# EPICS SNL sequencer program: timingApp/src/timingSequence.st
program timingSequence ("T=,P=EVG1:,R=")

// Macros
//  T: Timing system record prefix.
//  P:, R: Event generator record prefixes.
// Defaults provided here can be overridden by seq command in st.cmd.

// No wait for connections
option -c;
// Safe mode
option +s;
// Enable run-time debug messages
option +d;

#include "timingSequenceConstants.h"
%%#include <stdio.h>
%%#include <stdlib.h>

/*
 * Additional ticks for end of cycle
 */
int endOfCycleDelay;
assign endOfCycleDelay to "{T}TimCycleDelay";
monitor endOfCycleDelay;

/*
 * Injection request waveform.
 */
int request[7];
assign request to "{T}TimInjReq";
monitor request;
evflag requestFlag;
sync request requestFlag;
unsigned int modeIndexes[255];
%{
typedef enum { /* Request waveform indices. */
        TARGET_BUCKET,
        GUN_BUNCHES,
        INJ_MODE,
        GUN_INHIBIT,
        TARGET_AR_BUCKET,
        FUTURE_USE_1,
        SEQUENCE,
} REQUEST_FIELDS;
}%

/* Values extracted from injection request waveform: */
int sequence = 0;       /* Sequence #: request ignored if no change from previous */
int lastSequence = -1;
int bucket = 1;         /* Target bucket (1-328) */
int arBucket = 1;       /* AR Target bucket (1-304) */
assign arBucket to "{T}TimTargetARBucket";
int bunches = 1;        /* Number of electron gun bunches (1-16) */
int inhibit = 0;        /* Inhibit electron gun if set, even if mode allows gun */
int mode = 0;           /* Type of injection sequence.  See eventListForMode() */
int injFieldSync = 0;   /* Injection field delay */
int extrFieldSync = 0;  /* Extraction field delay */
int extrFieldARSync = 0;  /* Extraction field AR delay */
int extrFieldARSyncSP = 0;  /* Extraction field AR delay in AR/BR alignment cycles */
int brTgtBucket = 1;  /* BR target bucket (in buckets) for AR injection */

int injFieldSyncDelay = 0;
assign injFieldSyncDelay to "{T}TimInjFieldSyncDelay";
monitor injFieldSyncDelay;
int extrFieldSyncDelay = 0;
assign extrFieldSyncDelay to "{T}TimExtrFieldSyncDelay";
monitor extrFieldSyncDelay;
int extrFieldARSyncDelay = 0;
assign extrFieldARSyncDelay to "{T}TimExtrFieldARSyncDelay";
monitor extrFieldARSyncDelay;
int extrFieldARSyncDelaySP = 0;
assign extrFieldARSyncDelaySP to "{T}TimExtrFieldARSyncDelaySP";
monitor extrFieldARSyncDelaySP;
int injStBRBucket = 1;
assign injStBRBucket to "{P}{R}INJ:stBRBucket";
monitor injStBRBucket;

/* Save value until we're ready to write to the FPGA */
int injSyncMode;
assign injSyncMode to "{T}TimInjSyncMode";
int injAlignSel;
assign injAlignSel to "{T}TimInjAlignSel";

/*
 * Monitor of injection request values sent to FPGA sequencer.
 */

int sequenceMon = 0;        /* Sequence #: request ignored if no change from previous */
assign sequenceMon to "{T}TimSequenceNumberMon";
int bucketMon = 1;          /* Target bucket (1-328) */
assign bucketMon to "{T}TimTargetBucketMon";
int arBucketMon = 1;          /* Target AR Bucket (1-304) */
assign arBucketMon to "{T}TimTargetARBucketMon";
int bunchesMon = 1;         /* Number of electron gun bunches (1-16) */
assign bunchesMon to "{T}TimGunBunchCountMon";
int inhibitMon = 0;         /* Inhibit electron gun if set, even if mode allows gun */
assign inhibitMon to "{T}TimGunInhibitMon";
int modeMon = 0;            /* Type of injection sequence.  See eventListForMode() */
assign modeMon to "{T}TimInjModeMon";
int injFieldSyncMon = 0;    /* Injection field delay */
assign injFieldSyncMon to "{T}TimInjFieldSyncDelayMon";
int extrFieldSyncMon = 0;   /* Extraction field delay */
assign extrFieldSyncMon to "{T}TimExtrFieldSyncDelayMon";
int extrFieldARSyncMon = 0;   /* Extraction field delay */
assign extrFieldARSyncMon to "{T}TimExtrFieldARSyncDelayMon";

/*
 * Calculated values
 */
int injStBRBucketIdx = 0;

int tgtBRDelayOffset = 0;
assign tgtBRDelayOffset to "{T}TimTgtBRDelayOffset";
int tgtBRBucket = 1;
assign tgtBRBucket to "{T}TimTgtBRBucket";

/*
 * Storage ring current.
 * Sequencer refuses to inject when this exceeds MAX_BEAM_CURRENT.
 */
double beamcurrent;
assign beamcurrent to "SR:DCCT:AVG";
monitor beamcurrent;

/*
 * Soft sequence timestamp remainder which is used to set
 * the fine delay PV B0215:EVR1-Out:UDC0:Delay-SP .
 * D = 4 * S * R, where:
 * D is the fine delay setpoint value (10ps steps)
 * S is a scaling factor
 * R is the target bucket delay remainder
 * Initially, S can be set to 200, which will give precise 2ns steps
 *  for the possible values of the remainder:
 * R = [0, 0.25, 0.5, 0.75]
 * D = [0, 200, 400, 600]
 */

int boExtrDelay;
assign boExtrDelay to "B0215:EVR1-Out:UDC0:Delay-SP";

double boExtrDelayRemainder;
assign boExtrDelayRemainder to "B0215:TimSeqRemainder";

int boExtrDelayOffset;
assign boExtrDelayOffset to "B0215:TimSeqFineDelayOffst";
monitor boExtrDelayOffset;

int boExtrFineDelay;
assign boExtrFineDelay to "B0215:TimSeqFineDelay";

/*
 * lookup table which corespons to the remainder
 * {0, 0.25, 0.5, 0.75}
 */
#define BO_EXTR_FINE_DELAY_LT_SIZE  4
#define BO_EXTR_FINE_DELAY_STEP     200
int boExtrFineDelayLookupTable[BO_EXTR_FINE_DELAY_LT_SIZE] = {
    0*BO_EXTR_FINE_DELAY_STEP,
    1*BO_EXTR_FINE_DELAY_STEP,
    2*BO_EXTR_FINE_DELAY_STEP,
    3*BO_EXTR_FINE_DELAY_STEP};

/*
 * Overall timing system enable/disable
 */
int potentate;
assign potentate to "{T}TimPotentate";
monitor potentate;

/*
 * If set to 1, makes the FPGA generate the default sequence
 * if it doesn't receive a request within the alloted time slot
 */
int injCycleEnable;
assign injCycleEnable to "{P}{R}INJ:injCycleEnable";
monitor injCycleEnable;

/*
 * This request a single shot sequence and doesn't
 * make the FPGA generate any default sequence if
 * it doesn't receive a new request.
 */
int injSingleShot;
assign injSingleShot to "{P}{R}INJ:singleShot";

/*
 * Statistics
 */
%{
typedef enum {
    FC_SUCCESS,
    FC_MISSING_CONNECTION,
    FC_START_OVERRUN,
    FC_STALE_SEQUENCE,
    FC_INVALID_MODE,
    FC_INVALID_BUCKET,
    FC_INVALID_BUNCHES,
    FC_INVALID_BEAM_CURRENT,
    FC_EXCESSIVE_BEAM_CURRENT,
    FC_PV_SEVERITY,
    FC_BAD_EVR,
    FC_NO_EOS,
} FAULT_CODE;
}%
int goodCount;
assign goodCount to "{T}InjSeqSuccessCount";
int badCount;
assign badCount to "{T}InjSeqFailedCount";
int faultCode;
assign faultCode to "{T}InjSeqFaultCode";
int duplicateTimestampFound;
assign duplicateTimestampFound to "{T}InjSeqDupTimestamp";
int startOverrunCount;
assign startOverrunCount to "{T}InjSeqStartOverrunCount";

/*
 * Diagnostics
 */
int debugFlag;
assign debugFlag to "{T}InjSeqDebug";
monitor debugFlag;

/**
 * Mapping of # gun bunches to injection field trigger
 */
double bunchesToField[MAX_BUNCHES];
assign bunchesToField to "{T}GunBunchToInjFieldTrigger";
monitor bunchesToField;
int gunBunchesDelay;

/*
 * Injection cycles are initiated only when all EVR links are good.
 */
int allEVRvalid;
assign allEVRvalid to "{T}TimAllEVRvalid";
monitor allEVRvalid;

/*
 * Event generator FPGA
 */
#define EVG_SEQ_STATUS_ACTIVE 0x8
#define EVG_SEQ_STATUS_BUSY   0x10
int evgSequence[EVG_SEQUENCE_CAPACITY];
assign evgSequence to "{P}{R}E1:SEQ1";
int evgSeqEnable;
assign evgSeqEnable to "{P}{R}E1:SEQ1:enable";
int evgSeqStatus;
assign evgSeqStatus to "{P}{R}E1:seqStatus";
monitor evgSeqStatus;
int evgSequencerStarts;
assign evgSequencerStarts to "{P}{R}E1:seqStarts";
monitor evgSequencerStarts;
int evgSequencerCurrentStarts;

%{
/*
 * Comparison routine for qsort
 * Primary sort on time stamp (first word)
 * Secondary sort on event code (second word)
 * No sort on category code (third word)
 */
static int
tsCompare(const void *a, const void *b)
{
    const int *ap = a, *bp = b;
    int diff;
    if ((diff = ap[0] - bp[0]) == 0) {
        diff = ap[1] - bp[1];
    }
    return diff;
}

/*
 * Ensure monotonically increasing time stamps
 * and convert time stamps to delay and category
 * relative category (only the first in the group
 * has the delay)
 */
static int
monotonicSequence(int count, int *tstampsEventsAndCat)
{
    int i, idx;
    int ret = 1;
    int prev = -1;
    int prevCat = 0;

    for (i = 0, idx = 0; i < count; i++, idx += 3) {
        int this = tstampsEventsAndCat[idx];
        int thisCat = tstampsEventsAndCat[idx+2];
        if ((i < (count - 1)) && (tstampsEventsAndCat[idx+3] <= this)) {
            ret = 0;
            tstampsEventsAndCat[idx+3] = this + 1;
        }

        tstampsEventsAndCat[idx] = (this - prev) - 1;
        tstampsEventsAndCat[idx+2] = (thisCat - prevCat) != 0? thisCat : 0;
        prev = this;
        prevCat = thisCat;
    }

    return ret;
}

#define END_OF_SEQUENCE_TICKS (1<<30)
/*
 * approx. 1.35s
 */
#define DELAY_END             168740000
#include "TimingLookups.h"

}%

ss ssTiming {
    /*
     * Initial state
     * Set up some stuff
     */
    state start {
        when() {
            duplicateTimestampFound = 0;
            pvPut(duplicateTimestampFound);
            /* Operate in single shot mode only*/
            injCycleEnable = 0;
            pvPut(injCycleEnable, SYNC);
        } state await_connections
    }

    /*
     * Request default sequence
     */
    state default_sequence {
        entry {
            if(debugFlag) printf("State: default_sequence\n");
        }
        when() {
            mode = 0;
            injFieldSync = injFieldSyncDelay;
            extrFieldSync = extrFieldSyncDelay;
            extrFieldARSync = extrFieldARSyncDelay;
            extrFieldARSyncSP = extrFieldARSyncDelaySP;
            injStBRBucketIdx = (injStBRBucket <= 0)?  0 : injStBRBucket-1;
        } state create_requested_sequence
    }

    /*
     * Wait for connections to complete
     */
    state await_connections {
        int oldConnectCount;
        entry {
            if(debugFlag) printf("State: await_connections\n");
            oldConnectCount = -1;
        }

        when (injCycleEnable != 0) { } state inj_cycle_disable

        when (pvConnectCount() == pvAssignCount()) {
            if (faultCode == FC_MISSING_CONNECTION) {
                faultCode = FC_SUCCESS;
                pvPut(faultCode);
            }
        } state await_potentate

        when (delay(10) && (pvConnectCount() != oldConnectCount)) {
            oldConnectCount = pvConnectCount();
            printf("Timing Sequencer: %d/%d connected\n", pvConnectCount(),
                                                          pvAssignCount());
            if (faultCode == FC_SUCCESS) {
                faultCode = FC_MISSING_CONNECTION;
                pvPut(faultCode);
            }
        } state await_connections
    }

    /*
     * Wait for potentate
     */
    state await_potentate {
        entry {
            if(debugFlag) printf("State: await_potentate\n");
        }

        when (pvConnectCount() != pvAssignCount()) { } state missing_connection
        when (injCycleEnable != 0) { } state inj_cycle_disable
        when (potentate != 0) { } state await_precompletion
    }

    /*
     * Wait for injection cycles to be disabled. Only operate in
     * single shot
     */
    state inj_cycle_disable {
        entry {
            if(debugFlag) printf("State: inj_cycle_disable\n");
            /* Operate in single shot mode only*/
            injCycleEnable = 0;
            pvPut(injCycleEnable, SYNC);
        }

        when (pvConnectCount() != pvAssignCount()) { } state missing_connection
        when (potentate == 0) { } state await_potentate
        when () { } state await_precompletion
    }

    /*
     * Wait for injection cycle to start
     */
    state await_start {
        entry { if(debugFlag) printf("State: await_start\n"); }

        when (pvConnectCount() != pvAssignCount()) { } state missing_connection
        when (potentate == 0) { } state no_potentate
        when (injCycleEnable != 0) { } state inj_cycle_disable

        when (delay(TIMEOUT_AWAIT_START)) {
            /* EVG never started. Assume dead and try again */
        } state default_sequence

        when ((evgSeqStatus & EVG_SEQ_STATUS_ACTIVE) != 0) {
        } state await_precompletion
    }

    /*
     * Wait for injection cycle to reach precompletion point
     */
    state await_precompletion {
        entry { if(debugFlag) printf("State: await_precompletion\n"); }

        when (pvConnectCount() != pvAssignCount()) { } state missing_connection
        when (potentate == 0) { } state no_potentate
        when (injCycleEnable != 0) { } state inj_cycle_disable

        when (efTestAndClear(requestFlag)) {
            /* Ignore requests outside expected window */
        } state await_precompletion

        when (delay(TIMEOUT_AWAIT_PRECOMPLETION)) {
            /* EVG never finished. Assume dead and try again */
        } state default_sequence

        when ((evgSeqStatus & EVG_SEQ_STATUS_BUSY) == 0) {
            evgSequencerCurrentStarts = evgSequencerStarts;
        } state await_request
    }

    /*
     * Watch for injection request
     */
    state await_request {
        entry { if(debugFlag) printf("State: await_request\n"); }

        when (pvConnectCount() != pvAssignCount()) { } state missing_connection
        when (potentate == 0) { } state no_potentate
        when (injCycleEnable != 0) { } state inj_cycle_disable

        when (delay(REQUEST_WINDOW)) {
            /* No request, default cycle will be emitted */
        } state default_sequence

        when (evgSequencerStarts != evgSequencerCurrentStarts) {
            faultCode = FC_START_OVERRUN;
            startOverrunCount++;
            pvPut(startOverrunCount);
        } state increment_bad_count

        when (efTestAndClear(requestFlag)) {
            if (sequence == request[SEQUENCE]) {
                /* No request, or perhaps it was truncated */
                state default_sequence;
            }
            bucket   = request[TARGET_BUCKET];
            bunches  = request[GUN_BUNCHES];
            mode     = request[INJ_MODE];
            inhibit  = request[GUN_INHIBIT];
            arBucket = request[TARGET_AR_BUCKET];
            sequence = request[SEQUENCE];
            injFieldSync = injFieldSyncDelay;
            extrFieldSync = extrFieldSyncDelay;
            extrFieldARSync = extrFieldARSyncDelay;
            extrFieldARSyncSP = extrFieldARSyncDelaySP;
            injStBRBucketIdx = (injStBRBucket <= 0)?  0 : injStBRBucket-1;
        } state validate_request
    }

    /*
     * Transient sequential states to validate, prepare, and send sequence
     */
    state validate_request {
        entry { if(debugFlag) printf("State: validate_request\n"); }

        when (sequence == lastSequence) {
            faultCode = FC_STALE_SEQUENCE;
        } state increment_bad_count

        when ((bucket < MIN_BUCKETS) || (bucket > MAX_BUCKETS)) {
            faultCode = FC_INVALID_BUCKET;
        } state increment_bad_count

        when ((arBucket < MIN_AR_BUCKETS) || (arBucket > MAX_AR_BUCKETS)) {
            faultCode = FC_INVALID_BUCKET;
        } state increment_bad_count

        when ((bunches < MIN_BUNCHES) || (bunches > MAX_BUNCHES)) {
            faultCode = FC_INVALID_BUNCHES;
        } state increment_bad_count

        when () {
        } state check_beamcurrent
    }

    state check_beamcurrent {
        entry { if(debugFlag) printf("State: check_beamcurrent\n"); }

        when ((mode == SRINJECTION_MODE) && (pvSeverity(beamcurrent) == pvSevrINVALID)) {
            faultCode = FC_INVALID_BEAM_CURRENT;
        } state increment_bad_count

        when ((mode == SRINJECTION_MODE) && (beamcurrent > MAX_BEAM_CURRENT)) {
            faultCode = FC_EXCESSIVE_BEAM_CURRENT;
        } state increment_bad_count

        when () {
        } state check_severities
    }

    state check_severities {
        entry { if(debugFlag) printf("State: check_severities\n"); }

        when ((pvSeverity(evgSeqStatus) != pvSevrNONE)
            || (pvSeverity(evgSequencerStarts) != pvSevrNONE)) {
            faultCode = FC_PV_SEVERITY;
        } state increment_bad_count

        when () {
        } state check_links
    }

    state check_links {
        entry { if(debugFlag) printf("State: check_links\n"); }

        when ((pvStatus(allEVRvalid) != pvStatOK) || (allEVRvalid == 0)) {
            faultCode = FC_BAD_EVR;
        } state increment_bad_count

        when () {
        } state create_requested_sequence
    }

    /*
     * Create the new sequence
     */
    state create_requested_sequence {
        entry { if(debugFlag) printf("State: create_requested_sequence\n"); }

        when () {
            %%const unsigned char *e;
            int targetBucketDelayRaw = 125 * ((bucket * 21) % 328);
            int targetBucketDelay = targetBucketDelayRaw / 4;
            int targetBucketDelayRem = targetBucketDelayRaw % 4;
            int i, nTStamps;
            int highwater = 0;
            int foundEOS = 0;

            /*
             * Calculate fine delay for booster extraction kicker
             */
            boExtrFineDelay = boExtrFineDelayLookupTable[targetBucketDelayRem];

            /*
             * Calculate BR target bucket delay offset for AR injection
             */
            tgtBRDelayOffset = (18*(extrFieldARSyncSP % BR_H_NUMBER) % BR_H_NUMBER);

            /*
             * Get time stamp for each event and merge into common array
             */
            e = eventListForMode(mode);
            if (e == NULL) {
                faultCode = FC_INVALID_MODE;
                state increment_bad_count;
            }

            injSyncMode = injSyncForMode(mode);
            if (injSyncMode < 0) {
                faultCode = FC_INVALID_MODE;
                state increment_bad_count;
            }

            injAlignSel = injAlignSelForMode(mode);
            if (injAlignSel < 0) {
                faultCode = FC_INVALID_MODE;
                state increment_bad_count;
            }

            gunBunchesDelay = bunchesToField[bunches-1];
            memset(evgSequence, 0, sizeof(evgSequence[0])*EVG_SEQUENCE_CAPACITY);
            for (i = 0, nTStamps = 0; i < MAX_SEQUENCE_LENGTH; i++) {
                int event = e[i];
                int tstamp;
                int category;

                if (inhibit) {
                    if (event == GUNON_EVTCODE || event == GUNOFF_EVTCODE) {
                        continue;
                    }
                }

                if (event == SEQUENCE_END_EVTCODE) {
                    tstamp = DELAY_END + endOfCycleDelay;
                    category = 0;
                }
                else {
                    tstamp = getTimestamp(mode, event, injFieldSync, tgtBRDelayOffset, extrFieldSync,
                            extrFieldARSync, bunches, gunBunchesDelay, targetBucketDelay);
                    category = getCategory(mode, event);
                    if (tstamp > (END_OF_SEQUENCE_TICKS / 2)) {
                        tstamp = highwater + (tstamp - END_OF_SEQUENCE_TICKS) + 2;
                    }

                    if (tstamp < 0) {
                        fprintf(stderr, "WARNING: tstamp for evtcode %d is %d"
                                               " -- ignoring\n", event, tstamp);
                        continue;
                    }

                    if (category < 0) {
                        fprintf(stderr, "WARNING: category for evtcode %d is %d"
                                               " -- ignoring\n", event, category);
                        continue;
                    }

                    if (tstamp >= highwater) {
                        highwater = tstamp + 1;
                    }
                }

                evgSequence[(3*nTStamps)+0] = tstamp;
                evgSequence[(3*nTStamps)+1] = event;
                evgSequence[(3*nTStamps)+2] = category;
                nTStamps++;

                if (event == SEQUENCE_END_EVTCODE) {
                    foundEOS = 1;
                    break;
                }
            }

            if (!foundEOS) {
                faultCode = FC_NO_EOS;
                state increment_bad_count;
            }

            qsort(evgSequence, nTStamps, 3*sizeof(int), tsCompare);
            if (!monotonicSequence(nTStamps, evgSequence)) {
                duplicateTimestampFound = 1;
                pvPut(duplicateTimestampFound);
            }
        } state load_requested_sequence
    }

    state load_requested_sequence {
        entry {
            if(debugFlag) {
                printf("State: load_requested_sequence\n");
                if(debugFlag >= 2) {
                    int i;
                    for (i = 0 ; i < 7 ; i++) {
                        printf(" %d", request[i]);
                    }
                    printf("\n");
                }
            }
        }
        when (pvConnectCount() != pvAssignCount()) { } state missing_connection
        when (potentate == 0) { } state no_potentate
        when (injCycleEnable != 0) { } state inj_cycle_disable
        when (evgSequencerStarts != evgSequencerCurrentStarts) {
            faultCode = FC_START_OVERRUN;
            startOverrunCount++;
            pvPut(startOverrunCount);
        } state increment_bad_count

        when ((evgSeqStatus & EVG_SEQ_STATUS_ACTIVE) == 0) {

            pvPut(arBucket);
            pvPut(injAlignSel);
            pvPut(injSyncMode);

            pvPut(tgtBRDelayOffset);

            tgtBRBucket = ((injStBRBucketIdx +
                72*(extrFieldARSyncSP % BR_H_NUMBER)) % BR_H_NUMBER) + 1;
            pvPut(tgtBRBucket);

            pvPut(boExtrFineDelay);
            boExtrDelay = boExtrFineDelay + boExtrDelayOffset;
            pvPut(boExtrDelay);
            boExtrDelayRemainder = (double) boExtrFineDelay /
                BO_EXTR_FINE_DELAY_STEP / BO_EXTR_FINE_DELAY_LT_SIZE;
            pvPut(boExtrDelayRemainder);

            pvPut(evgSequence);
            evgSeqEnable = 1;
            pvPut(evgSeqEnable);
            injSingleShot = 1;
            pvPut(injSingleShot);
            lastSequence = sequence;
            faultCode = FC_SUCCESS;
            pvPut(faultCode);
            goodCount++;
            pvPut(goodCount);

            /* assign monitor values to injection parameters */
            sequenceMon = sequence;
            pvPut(sequenceMon);
            bucketMon = bucket;
            pvPut(bucketMon);
            bunchesMon = bunches;
            pvPut(bunchesMon);
            inhibitMon = inhibit;
            pvPut(inhibitMon);
            arBucketMon = arBucket;
            pvPut(arBucketMon);
            modeMon = mode;
            pvPut(modeMon);
            injFieldSyncMon = injFieldSync;
            pvPut(injFieldSyncMon);
            extrFieldSyncMon = extrFieldSync;
            pvPut(extrFieldSyncMon);
            extrFieldARSyncMon = extrFieldARSync;
            pvPut(extrFieldARSyncMon);
        } state await_start
    }

    state no_potentate {
        when() {
            injCycleEnable = 0;
            pvPut(injCycleEnable, SYNC);
        } state await_potentate
    }

    state missing_connection {
        when() {
            faultCode = FC_MISSING_CONNECTION;
            pvPut(faultCode);
            injCycleEnable = 0;
            pvPut(injCycleEnable, SYNC);
        } state await_connections
    }

    state increment_bad_count {
        entry { if(debugFlag) printf("State: increment_bad_count\n"); }
        when() {
            pvPut(faultCode);
            badCount++;
            pvPut(badCount);
        } state await_precompletion
    }
}
